Universal Robots PolyScope program: ad_lab_exe_3_4_52.urp

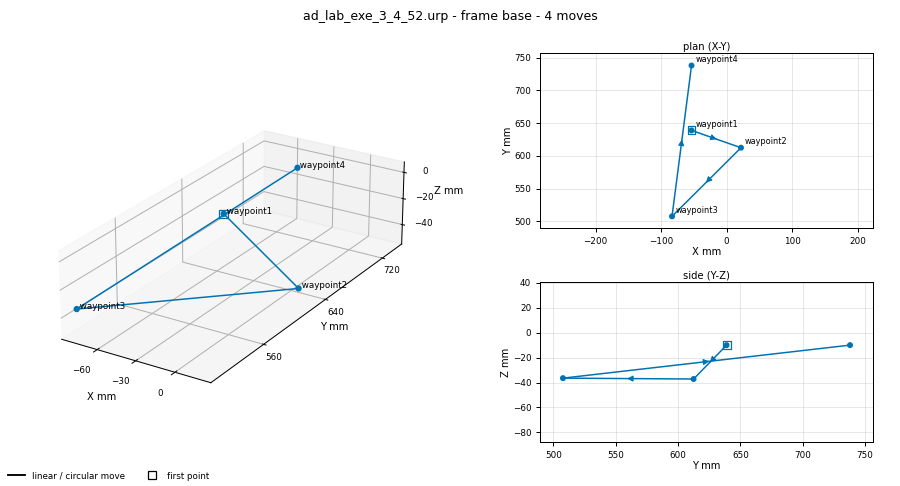
[picture p0: tool path of ad_lab_exe_3_4_52.urp in frame base, 4 of 4 moves have a stored position in this frame; points joined in program order, loops and branches not executed]
Program ad_lab_exe_3_4_52 (createdIn=3.2.19293 lastSavedIn=3.2.19293 directory=/programs installation=default robotSerialNumber=2015351391)
Calibrated DH parameters: a=[0.000352, -0.161198, -0.373486, 0.00005, 0.000049, 0]; d=[0.089268, 352.477598, -320.08558, -32.281492, 0.094939, 0.082518]; alpha=[1.570728, 0.001116, -0.003686, 1.571189, -1.570572, 0]; deltaTheta=[-0.000012, 1.181849, -1.491165, 0.309495, -0.000007, 0.000025]
Robot Program (runOnlyOnce=false motionType=MoveJ speed=1.047198 acceleration=1.396263 recalculateMotions=false)
  MoveL speed 250 mm/s, acceleration 2500 mm/s^2 (recalculateMotions=false) feature(featureName=plane_2)
    Waypoint waypoint1: TCP in base x=-53.573 y=638.899 z=-10.031 mm, rx=-2.2353 ry=-2.1151 rz=-0.1037 rad; joints [105.373, -122.001, -99.762, -43.28, 88.161, -71.757] deg; pose in feature x=8.79 y=-0.006 z=-99.576 mm, rx=-0.001 ry=0.004 rz=-0.0006 rad; flange x=-54.33 y=627.452 z=114.458 mm, rx=-2.2354 ry=-2.115 rz=-0.1037 rad
    Waypoint waypoint2: TCP in base x=21.961 y=612.434 z=-37.197 mm, rx=-2.3554 ry=-1.9983 rz=-0.1175 rad; joints [99.194, -121.815, -105.605, -37.866, 87.666, -71.754] deg; pose in feature x=-15.714 y=76.891 z=-74.474 mm, rx=-0.0204 ry=0.0023 rz=0.1069 rad; flange x=18.805 y=601.457 z=87.256 mm, rx=-2.3554 ry=-1.9984 rz=-0.1175 rad
    Waypoint waypoint3: TCP in base x=-83.379 y=507.599 z=-36.492 mm, rx=-2.1407 ry=-2.2468 rz=0.0157 rad; joints [111.228, -112.926, -119.947, -35.42, 91.351, -71.75] deg; pose in feature x=-125.778 y=-22.434 z=-84.862 mm, rx=0.0391 ry=-0.0689 rz=-0.1026 rad; flange x=-79.06 y=505.221 z=88.407 mm, rx=-2.1407 ry=-2.2468 rz=0.0157 rad
    Waypoint waypoint4: TCP in base x=-53.573 y=738 z=-9.993 mm, rx=-2.2335 ry=-2.1123 rz=-2.1123 rad; joints [103.268, -132.699, -80.302, -51.764, 88.307, -73.823] deg; pose in feature x=107.359 y=-5.537 z=-90.932 mm, rx=-1.2512 ry=0.3431 rz=-0.0551 rad; flange x=68.819 y=384.862 z=62.446 mm, rx=-2.4339 ry=-1.962 rz=0.0087 rad
